// TIA Portal V18 export
// export: Created 2026-01-09T11:23:23.7986929Z, ExportSetting WithDefaults, DisplayName Totally Integrated Automation Portal, DisplayVersion V18 Update 5, DisplayName TIA Portal Openness, DisplayVersion V18 Update 5, DisplayName TIA Portal Teamcenter Gateway, DisplayVersion V18, DisplayName TIA Portal Version Control Interface, DisplayVersion V18, DisplayName SINAMICS Startdrive Advanced, DisplayVersion V18 SP2 Update 1, DisplayName SINAMICS Startdrive G110M, G120, G120C, G120D, G120P, G115D, DisplayVersion V18 SP2 Update 1, DisplayName SINAMICS Startdrive G130, G150, S120, S150, SINAMICS MV, S210, G220, S200, DisplayVersion V18 SP2 Update 1, DisplayName STEP 7 Professional, DisplayVersion V18 Update 5, DisplayName STEP 7 Safety, DisplayVersion V18, DisplayName WinCC Professional, DisplayVersion V18 Update 5
Screen "GMT"  1280x800, Number=4, Template=11GMT
  on GenerateScreen: Loading(); SetBit(Tag := NormalON); ResetBit(Tag := NormalOFF); VBCom(Index := 5); LoadIO(); IOVisual(Funcode := 100, SubFuncode := 0); LoadCylinder()
  ScreenLayer 
    GraphicView "图形视图_1" at 284,599 size 430x85  Picture=3c0f3e524cdb2dbf460d5f91a019f56
    TextField "文本域_4" at 136,222 size 577x35  Text="浙江金麦特集团有限公司 / Headquarters: Zhejiang GMT Group Co., Ltd. / Zhejiang Jinmaite Group Co., Ltd."
    TextField "文本域_6" at 136,435 size 631x27  Text="https://www.goldmt.net/index.aspx"
    TextField "文本域_2" at 136,266 size 1401x62  Text="浙江省长兴县经济开发区发展大道399号 After Service:+(86)-(0572)-6297-522 / 399 Development Avenue, Economic Development Zone, Changxing County, Zhejiang ProvinceAfter Service: +(86)-(0572)-6297-522 / č. 399, Development Avenue, ekonomická rozvojová zóna, Changxing, provincie Zhejiang Po servise:+(86)-(0572)-6297-522"
    TextField "文本域_3" at 136,351 size 1141x62  Text="No. 399 Development Avenue, Economic Development Zone, Changxing County, Zhejiang Province Innovation Leads the Way in Technology; Intelligence Shapes the Future / Č. 399 Development Avenue, Zóna hospodárskeho rozvoja, okres Changxing, provincia Zhejiang Inovácie vedú cestu v technológii; inteligencia formuje budúcnosť"
    SymbolicIOField "seaText1" at 131,72 size 1146x65  CountVisibleItems=3, Mode=Output, OnValue=1, StyleItem=sltDeepBold22, TextList=XXXXX_PanelTextlist, TextOff="0", TextOn="1"
      ProcessValue := Sys_VersionManagement_HMIPageID
    Button "btnMenu1_2" at 0,230 size 128x75  Mode=Text, PictureOff=SS_00_000_HomeSmall, StyleItem=BtnActive18, TextOff="金麦特 / GMT"
      on Release: ActivateScreen(Screen name := , Object number := 0); SetTag(Tag := Sys_VersionManagement_HMIPageID, Value := 4)
    TextField "Template_Text field_1" at 855,4 size 299x25  Text="Tool scanning code is running"
      RangeAppearanceAnimation "RangeAppearanceAnimation"
        tag ChangeOver_DB_Global_ScanFixtureFlag
        1..1: back #00ff00, fore #31344a, flashing
      SingleBitVisibilityAnimation "VisibilityAnimation"
        tag ChangeOver_DB_Global_ScanFixtureFlag
